KUKA KRL data list: AMM_USER.dat

&ACCESS RV
&REL 1
&COMMENT KEB Milling User Interface
&USER UTEC
&PARAM EDITMASK = *
&PARAM TEMPLATE = C:\KRC\Roboter\Template\ExpertVorgabe
DEFDAT AMM_user PUBLIC



ENDDAT
